{attribute 'linkalways'} 
{attribute 'no_explicit_call' := 'This FB is a CLASS and must be accessed using methods or properties'}
{attribute 'enable_dynamic_creation'}
FUNCTION_BLOCK Node_F_VN_EnclosingRectangle EXTENDS VisionNode
VAR
    ipPointSet : _ITcVnContainer;
    stRectangle : _TcVnRotatedRectangle;
    hrPrev : _HRESULT(S_OK);
	hresult : _HRESULT(S_OK);
END_VAR

METHOD PUBLIC  Clone : I_Node
VAR
	pNode : POINTER TO Node_F_VN_EnclosingRectangle;
END_VAR
pNode := __NEW(Node_F_VN_EnclosingRectangle);
Clone := pNode^;
END_METHOD

METHOD FB_init : BOOL
VAR_INPUT
	bInitRetains : BOOL; // if TRUE, the retain variables are initialized (warm start / cold start)
	bInCopyCode : BOOL;  // if TRUE, the instance afterwards gets moved into the copy code (online change)
END_VAR
AddInput('ipPointSet', ipPointSet);
AddInput('hrPrev', hrPrev);
AddOutput('stRectangle', stRectangle);
AddOutput('hresult',hresult);
END_METHOD

METHOD PROTECTED OnExecute
hresult.Value := F_VN_EnclosingRectangle(
	ipPointSet := ipPointSet.Value,
    stRectangle := stRectangle.Value,
	hrPrev:= hrPrev.Value);
END_METHOD

METHOD PUBLIC PreExecutionCheck
VAR_INPUT
	Check : I_PreExecutionChecks;
END_VAR
Check.IsTrue(ipPointSet.IsValid, 'ipPointSet must be a valid container');
Check.IsTrue((ipPointSet.IsType(TC_GLOBAL_CONST_LIST.ContainerType_Vector_TcVnPoint2_DINT) OR
              ipPointSet.IsType(TC_GLOBAL_CONST_LIST.ContainerType_Vector_TcVnPoint2_REAL)),
              'ipPointSet contains incorrect type');
END_METHOD

END_FUNCTION_BLOCK

(* stored: Version 1.1.0.1, ProductVersion 3.1.4026.13
   POU Node_F_VN_EnclosingRectangle: Id {c4a4e0ef-a465-0dd1-2553-5b4da54e0837}, SpecialFunc None
   Folder Constructor: Id {8583cf63-0e82-0e40-19ba-f93036e91daf}
   Method Clone: Id {edaf76a4-1cde-0b40-27ca-105259c99552}
   Method FB_init: Id {ff8094c3-0021-0814-2dff-cb7c16322efd}
   Method OnExecute: Id {0b220b9c-be71-0408-2abf-9ba747e48e79}
   Method PreExecutionCheck: Id {2536ff90-27c4-0d53-238a-235012985046} *)
